// TIA Portal V19 export
TYPE "Positioning_MOL_Machine_DataOut"
// stored: Access Published
   STRUCT
      M_Contactor_Minus : Bool;
      M_Contactor_Plus : Bool;
   END_STRUCT;
END_TYPE
